// TwinCAT 3 PLC project ExceptionTest
// ProgramVersion: 3.1.4023.0
// libraries:
//   Tc2_Standard, * (Beckhoff Automation GmbH)
//   Tc2_System, * (Beckhoff Automation GmbH)
//   Tc2_Utilities, * (Beckhoff Automation GmbH)
//   Tc3_Module, * (Beckhoff Automation GmbH)
// project tree:
//   DUTs/ E_Exception.TcDUT, E_Origin.TcDUT, E_Signal.TcDUT, ST_Exception.TcDUT, ST_Signal.TcDUT
//   / PlcTask.TcTTO
//   POUs/ Catch.TcPOU, ExceptionHandling.TcPOU, HigherLevelFB.TcPOU, I_ExceptionHandling.TcIO, I_SignalHandling.TcIO, MAIN.TcPOU, SignalHandling.TcPOU, System.TcPOU, TestFB.TcPOU, Try.TcPOU
// real-time tasks:
//   TASK PlcTask: cycle T#10ms, priority 20, ADS port 350

CONFIGURATION ExceptionTest
    RESOURCE PLC ON TwinCAT3
        TASK PlcTask(INTERVAL := T#10ms, PRIORITY := 20);
        PROGRAM MAIN WITH PlcTask : MAIN;
    END_RESOURCE
END_CONFIGURATION

// ---- DUTs/E_Exception.TcDUT

TYPE E_Exception :
(
	eNO_EXCEPTION := 0,
	eWRONG_VALUE_EXCEPTION := 100,
	eLOW_PRESSURE_EXCEPTION := 110,
	eSYSTEM_EXCEPTION := 10000
);
END_TYPE

// ---- DUTs/E_Origin.TcDUT
 TYPE E_Origin :
(
	eNO_ORIGIN := 0,
	eTEST_UNIT := 100,
	eHIGHER_LEVEL := 110
);
END_TYPE

// ---- DUTs/E_Signal.TcDUT
TYPE E_Signal :
(
	eNO_SIGNAL := 0,
	eWAIT_FOR_RELEASE_SIGNAL := 100
);
END_TYPE

// ---- DUTs/ST_Exception.TcDUT
TYPE ST_Exception :
STRUCT
	eException : E_Exception;
	eExceptionOrigin : E_Origin;
	sTimestamp : STRING;
END_STRUCT
END_TYPE

// ---- DUTs/ST_Signal.TcDUT
TYPE ST_Signal :
STRUCT
	eSignal : E_Signal;
	eSignalOrigin : E_Origin;
	sTimestamp : STRING;
END_STRUCT
END_TYPE

// ---- POUs/I_ExceptionHandling.TcIO
INTERFACE I_ExceptionHandling

METHOD BuildException : ST_Exception
VAR_INPUT
	eException : E_Exception;
END_VAR
END_METHOD

METHOD Catch : BOOL
VAR_INPUT
	eException : E_Exception;
	eExceptionOrigin : E_Origin;
END_VAR
END_METHOD

METHOD ExceptionAvailable : BOOL
VAR_INPUT
END_VAR
END_METHOD

METHOD ForwardToNextLevel : BOOL
VAR_INPUT
	sender : I_ExceptionHandling;
END_VAR
END_METHOD

METHOD GenericCatch : BOOL
VAR_INPUT
	eException : E_Exception;
END_VAR
END_METHOD

PROPERTY getException : ST_Exception
GET
END_GET
END_PROPERTY

PROPERTY getExceptionOrigin : E_Origin
GET
END_GET
END_PROPERTY

METHOD Throw : BOOL
VAR_INPUT
	stException : ST_Exception;
END_VAR
END_METHOD

END_INTERFACE

// ---- POUs/I_SignalHandling.TcIO
INTERFACE I_SignalHandling

METHOD BuildSignal : ST_Signal
VAR_INPUT
	eSignal	: E_Signal;
END_VAR
END_METHOD

METHOD GenericReceive : BOOL
VAR_INPUT
	eSignal : E_Signal;
END_VAR
END_METHOD

PROPERTY getSignal : ST_Signal
GET
END_GET
END_PROPERTY

PROPERTY getSignalOrigin : E_Origin
GET
END_GET
END_PROPERTY

METHOD GlobalReset 
VAR_INPUT
END_VAR
END_METHOD

METHOD Receive : BOOL
VAR_INPUT
	eSignal : E_Signal;
	eSignalOrigin : E_Origin;
END_VAR
END_METHOD

METHOD ResetSignal : BOOL
VAR_INPUT
	eSignal : E_Signal;
	eSignalOrigin : E_Origin;
END_VAR
END_METHOD

METHOD Signal : BOOL
VAR_INPUT
	stSignal	: ST_Signal;
END_VAR
END_METHOD

METHOD SignalAvailable : BOOL
VAR_INPUT
END_VAR
END_METHOD

END_INTERFACE

// ---- POUs/MAIN.TcPOU
PROGRAM MAIN
VAR
	fbHigherLevel : HigherLevelFB;
	eException : E_Exception;
	stException : ST_Exception;
	
	bSystemException : BOOL;
	bLowPressureException : BOOL;
	bTestUnitWaitingForRelease : BOOL;
END_VAR

fbHigherLevel(eOrigin := eHIGHER_LEVEL);

IF fbHigherLevel.Receive(eWAIT_FOR_RELEASE_SIGNAL, eTEST_UNIT) 
THEN
	bTestUnitWaitingForRelease := TRUE;
END_IF

WHILE fbHigherLevel.ExceptionAvailable()
DO

	stException := fbHigherLevel.getException;
	
	CASE stException.eException OF
	
		eSYSTEM_EXCEPTION:
			//Stop machine operation for example
			bSystemException := TRUE;
			;
		eLOW_PRESSURE_EXCEPTION:
			bLowPressureException := TRUE;
			;
			
	END_CASE
	
END_WHILE

END_PROGRAM

// ---- POUs/HigherLevelFB.TcPOU
FUNCTION_BLOCK HigherLevelFB EXTENDS SignalHandling
VAR_INPUT
END_VAR
VAR_OUTPUT
END_VAR
VAR
	fbTest : TESTFB;
	stException : ST_Exception;
	bSystemException : BOOL;
	bWrongValueException : BOOL;
END_VAR

SUPER^();
fbTest(eOrigin := eTEST_UNIT);

IF fbTest.Catch(eWRONG_VALUE_EXCEPTION, fbTest.getExceptionOrigin) 
THEN
	;
// React to error here
// Catch must reset the exception in fbTest
	bWrongValueException := TRUE;	
END_IF

//Forward all other exceptions to the next higher level
IF fbTest.ExceptionAvailable()
THEN

	//ForwardToNextLevel must set all exceptions in fbTest on forwarded
	ForwardToNextLevel(fbTest);
	
END_IF

IF bSystemException
THEN
	Throw(BuildException(eSYSTEM_EXCEPTION));
END_IF

END_FUNCTION_BLOCK

// ---- POUs/SignalHandling.TcPOU
(*
Signals are sent only once.
In order to resend the same signal, a global or a local reset is necessary.
*)
FUNCTION_BLOCK SignalHandling EXTENDS ExceptionHandling IMPLEMENTS I_SignalHandling 
VAR_OUTPUT
END_VAR

VAR_STAT
	bResetSignals : BOOL;
	aSignals : ARRAY[1..cMaxNumSignals] OF ST_Signal;
	uiSignalCounter : UINT := 0;
END_VAR

VAR CONSTANT
	cMaxNumSignals : UINT := 200;
	aEmptySignals : ARRAY[1..cMaxNumSignals] OF ST_Signal;
END_VAR

SUPER^();

METHOD BuildSignal : ST_Signal
VAR_INPUT
	eSignal	: E_Signal;
END_VAR
BuildSignal.eSignal := eSignal;
BuildSignal.eSignalOrigin := getSignalOrigin;
BuildSignal.sTimestamp := SYSTEMTIME_TO_STRING(fbTime.systemTime);
END_METHOD

METHOD GenericReceive : BOOL
VAR_INPUT
	eSignal : E_Signal;
END_VAR
VAR
	i : UINT;
END_VAR
FOR i := 1 TO uiSignalCounter
DO

	IF aSignals[i].eSignal = eSignal
	THEN
		//Reset the signal now
		GenericReceive := TRUE;
		RETURN;
	END_IF
		
END_FOR
END_METHOD

{warning 'Eigenschaftenimplementierung hinzufügen'}
PROPERTY getSignal : ST_Signal
GET
VAR CONSTANT
	stEmptySignal : ST_Signal;
END_VAR
IF SignalAvailable()
THEN
	getSignal := aSignals[uiSignalCounter];
	aSignals[uiSignalCounter] := stEmptySignal;
	uiSignalCounter := uiSignalCounter - 1;
END_IF
END_GET
END_PROPERTY

PROPERTY getSignalOrigin : E_Origin
GET
getSignalOrigin := eOrigin;
END_GET
END_PROPERTY

METHOD GlobalReset 
VAR
	stEmptySignal : ST_Signal;
	i : UINT;
END_VAR
aSignals := aEmptySignals;
uiSignalCounter := 0;
END_METHOD

METHOD Receive : BOOL
VAR_INPUT
	eSignal : E_Signal;
	eSignalOrigin : E_Origin;
END_VAR
VAR
	i : UINT;
END_VAR
FOR i := 1 TO uiSignalCounter
DO

	IF aSignals[i].eSignal = eSignal
	AND_THEN aSignals[i].eSignalOrigin = eSignalOrigin
	THEN
		//Reset the signal now
		Receive := TRUE;
		RETURN;
	END_IF
		
END_FOR
END_METHOD

METHOD ResetSignal : BOOL
VAR_INPUT
	eSignal : E_Signal;
	eSignalOrigin : E_Origin;
END_VAR
VAR
	i , k: UINT;
	stEmptySignal : ST_Signal;
END_VAR
IF SignalAvailable()
THEN
	
	FOR i:= 1 TO uiSignalCounter 
	DO
		//Search for exception
		IF aSignals[i].eSignal = eSignal 
		AND_THEN aSignals[i].eSignalOrigin = eSignalOrigin
		THEN
			//If found delete it from the array and adjust it
			ResetSignal := TRUE;
			FOR k:= i TO uiSignalCounter-1
			DO
				aSignals[k] := aSignals[k+1];
			END_FOR
			aSignals[k+1] := stEmptySignal;
			uiSignalCounter := uiSignalCounter - 1;
		END_IF  
	END_FOR

END_IF
END_METHOD

METHOD Signal : BOOL
VAR_INPUT
	stSignal	: ST_Signal;
END_VAR
VAR
	i : UINT;
END_VAR
IF uiSignalCounter <= cMaxNumSignals
THEN
	//Check if signal has been already sent
	FOR i := 1 TO uiSignalCounter
	DO
	
		IF aSignals[i].eSignal = stSignal.eSignal
		AND_THEN aSignals[i].eSignalOrigin = stSignal.eSignalOrigin
		THEN
			RETURN;
		END_IF
			
	END_FOR
	
	uiSignalCounter := uiSignalCounter + 1;
	aSignals[uiSignalCounter] := stSignal;
	Signal := TRUE;
	
ELSE

	Signal := FALSE;
	
END_IF
END_METHOD

METHOD SignalAvailable : BOOL
SignalAvailable := uiSignalCounter > 0;
END_METHOD

END_FUNCTION_BLOCK

// ---- POUs/ExceptionHandling.TcPOU
FUNCTION_BLOCK ExceptionHandling EXTENDS System IMPLEMENTS I_ExceptionHandling

VAR_OUTPUT
END_VAR
VAR
	{attribute 'hide'} 
	uiExceptionCounter : UINT := 0;
	uiPresentExceptions : UINT := 0;
	aExceptions : ARRAY[1..cMaxNumExceptions] OF ST_Exception;
	
	
	
END_VAR

VAR CONSTANT
	cMaxNumExceptions : UINT := 200;
	aEmptyExceptions : ARRAY[1..cMaxNumExceptions] OF ST_Exception;
END_VAR

SUPER^();

aExceptions := aEmptyExceptions;

uiExceptionCounter := 0;
uiPresentExceptions := 0;


METHOD BuildException : ST_Exception
VAR_INPUT
	eException	: E_Exception;
END_VAR
BuildException.eException := eException;
BuildException.eExceptionOrigin := getExceptionOrigin;
BuildException.sTimestamp := SYSTEMTIME_TO_STRING(fbTime.systemTime);
END_METHOD


METHOD Catch : BOOL
VAR_INPUT
	eException : E_Exception;
	eExceptionOrigin : E_Origin;
END_VAR

VAR

	i,k : UINT;
	stEmptyException : ST_Exception;
END_VAR
IF ExceptionAvailable()
THEN
	
	FOR i:= 1 TO uiExceptionCounter 
	DO
		//Search for exception
		IF aExceptions[i].eException = eException 
		AND_THEN aExceptions[i].eExceptionOrigin = eExceptionOrigin
		THEN
			//If found delete it from the array and adjust it
			Catch := TRUE;
			FOR k:= i TO uiExceptionCounter-1
			DO
				aExceptions[k] := aExceptions[k+1];
			END_FOR
			aExceptions[k+1] := stEmptyException;
			uiExceptionCounter := uiExceptionCounter - 1;
		END_IF  
	END_FOR

END_IF
END_METHOD

METHOD ExceptionAvailable : BOOL
ExceptionAvailable := uiExceptionCounter > 0;
END_METHOD

METHOD ForwardToNextLevel : BOOL
VAR_INPUT
	sender	: I_ExceptionHandling;
END_VAR
WHILE sender.ExceptionAvailable()
DO

	//Report to next level
	Throw(sender.getException);
	
END_WHILE
END_METHOD

METHOD GenericCatch : BOOL
VAR_INPUT
	eException	: E_Exception;
END_VAR
VAR
	i,k : UINT;
	stEmptyException : ST_Exception;
END_VAR
IF ExceptionAvailable()
THEN
	
	FOR i:= 1 TO uiExceptionCounter 
	DO
		//Search for exception
		IF aExceptions[i].eException = eException 
		THEN
			//If found delete it from the array and adjust it
			GenericCatch := TRUE;
			FOR k:= i TO uiExceptionCounter-1
			DO
				aExceptions[k] := aExceptions[k+1];
			END_FOR
			aExceptions[k+1] := stEmptyException;
			uiExceptionCounter := uiExceptionCounter - 1;
		END_IF  
	END_FOR

END_IF
END_METHOD

PROPERTY getException : ST_Exception
GET
IF ExceptionAvailable()
THEN
	getException := aExceptions[uiExceptionCounter];
	uiExceptionCounter := uiExceptionCounter - 1;
END_IF
END_GET
END_PROPERTY

PROPERTY getExceptionOrigin : E_Origin
GET
getExceptionOrigin := eOrigin;
END_GET
END_PROPERTY

METHOD Throw : BOOL
VAR_INPUT
	stException	: ST_Exception;
END_VAR
IF uiExceptionCounter <= cMaxNumExceptions
THEN
	uiExceptionCounter := uiExceptionCounter + 1;
	aExceptions[uiExceptionCounter] := stException;
	Throw := TRUE;
ELSE
	Throw := FALSE;
END_IF

uiPresentExceptions := uiExceptionCounter;
END_METHOD

END_FUNCTION_BLOCK

// ---- POUs/System.TcPOU
FUNCTION_BLOCK System
VAR_INPUT CONSTANT
	eOrigin : E_Origin;
END_VAR
VAR_OUTPUT
END_VAR
VAR
	fbTime : FB_LocalSystemTime := ( bEnable := TRUE, dwCycle := 1 );
END_VAR

fbTime();

END_FUNCTION_BLOCK

// ---- POUs/Catch.TcPOU
FUNCTION Catch : BOOL
VAR_INPUT
	eException : E_Exception;
END_VAR
VAR_OUTPUT
END_VAR
VAR
END_VAR

END_FUNCTION

// ---- POUs/TestFB.TcPOU
FUNCTION_BLOCK TestFB EXTENDS SignalHandling
VAR_INPUT
	rTemperature : REAL;
END_VAR
VAR_OUTPUT
END_VAR
VAR
	bLowPressure : BOOL;
	bWaitForRelease : BOOL;
END_VAR

SUPER^();

IF rTemperature = 0 
THEN
	Throw(BuildException(eWRONG_VALUE_EXCEPTION));	
END_IF

IF bLowPressure
THEN
	Throw(BuildException(eLOW_PRESSURE_EXCEPTION));
END_IF

IF bWaitForRelease
THEN
	bWaitForRelease := FALSE;
	Signal(BuildSignal(eWAIT_FOR_RELEASE_SIGNAL));
END_IF

END_FUNCTION_BLOCK

// ---- POUs/Try.TcPOU
FUNCTION Try : BOOL
VAR_INPUT
	iExceptionHandling : I_ExceptionHandling;
END_VAR
VAR_OUTPUT
END_VAR
VAR
END_VAR

END_FUNCTION
